FUNCTION_BLOCK FB_System_BWK_931
VAR_INPUT
	Freigabe_auto			: BOOL;
	Betrieb_Anford_auto		: BOOL;
	Regelung_Sollw_auto		: REAL;
END_VAR
VAR_OUTPUT
	{attribute 'OPC.UA.DA' := '1'}Steuerung				: ST_System_BWK_Steuerung;		
	{attribute 'OPC.UA.DA' := '1'}Stellwert				: ST_System_BWK_Stellwert;		
	{attribute 'OPC.UA.DA' := '1'}Zustand					: ST_System_BWK_Zustand;	
	{attribute 'OPC.UA.DA' := '1'}Parameter				: ST_System_BWK_Parameter;		
END_VAR
VAR
	Stellventil_331			: FB_SV;
	Regelventil_331			: FB_RV;
	Brennwertkessel_931		: FB_BWK;

	Zustandscheck			: FB_System_BWK_Zustandscheck;
	Logik					: FB_System_BWK_Logik;
	Ablaufsteuerung			: FB_System_BWK_Ablaufsteuerung;
	Sollwertscheck			: FB_System_BWK_Sollwertscheck;
END_VAR
VAR // added by the converter: edge detectors and wires of the graphical bodies
    _w1, _w2 : ANY;
END_VAR

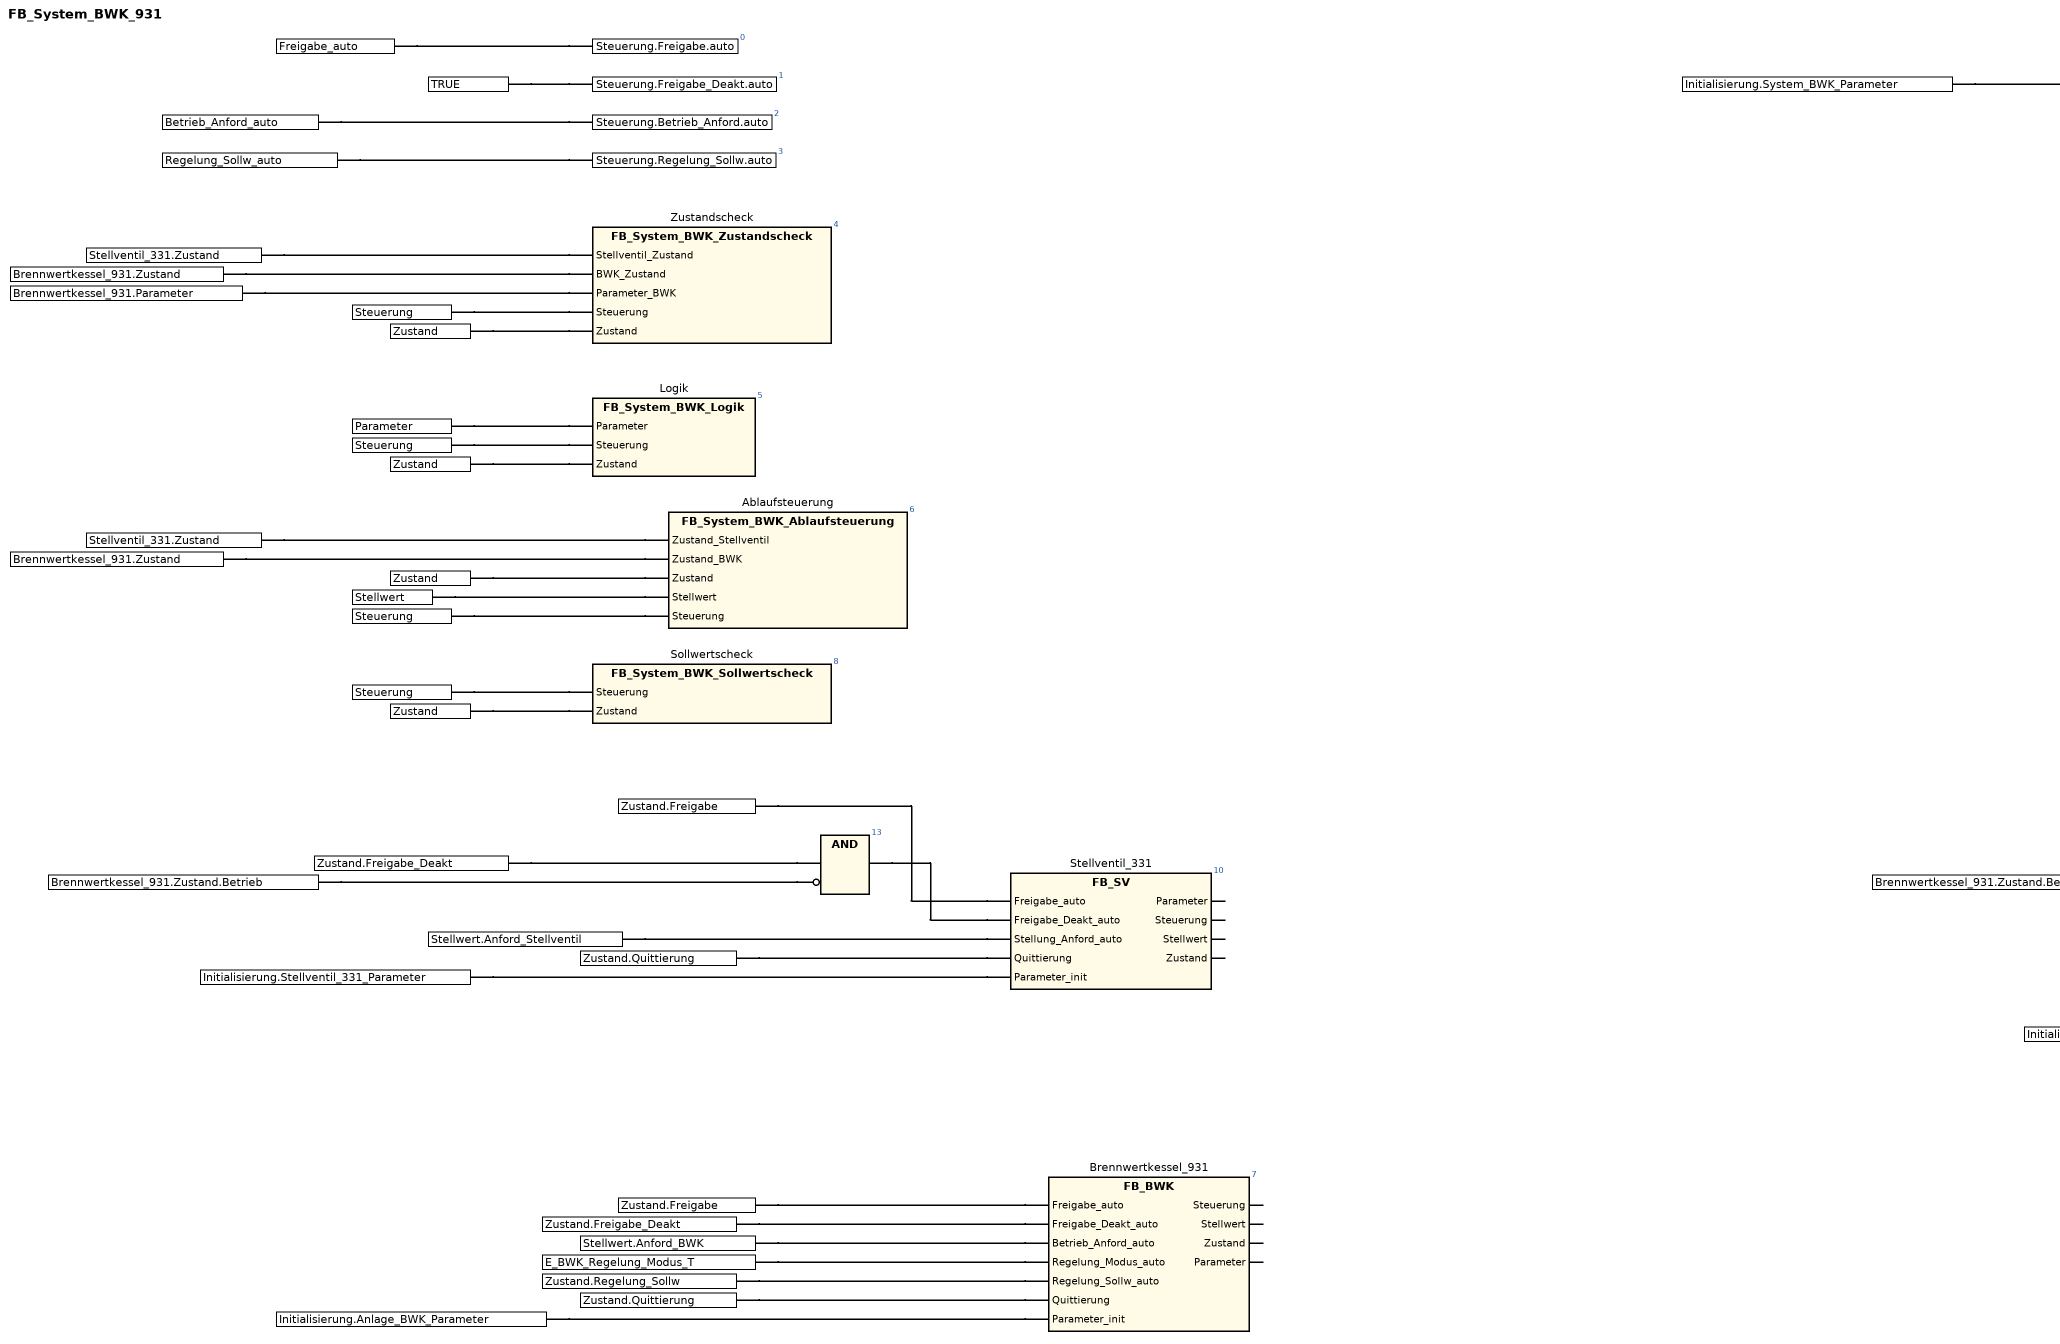
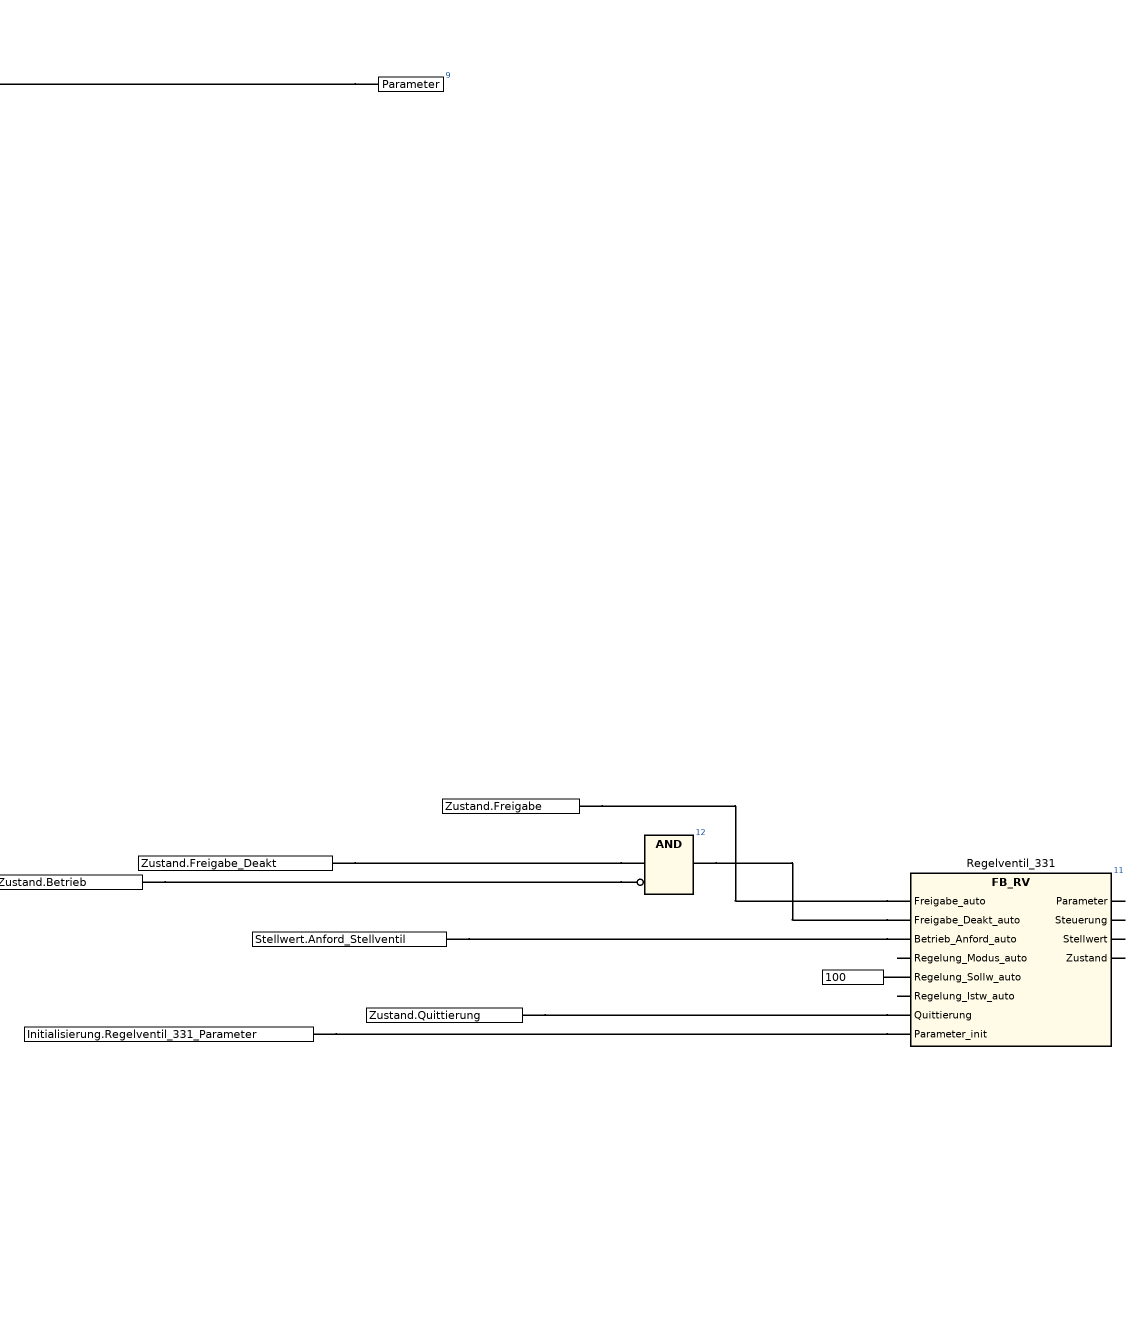
Steuerung.Freigabe.auto := Freigabe_auto;
Steuerung.Freigabe_Deakt.auto := TRUE;
Steuerung.Betrieb_Anford.auto := Betrieb_Anford_auto;
Steuerung.Regelung_Sollw.auto := Regelung_Sollw_auto;
Zustandscheck(
    Stellventil_Zustand := Stellventil_331.Zustand,
    BWK_Zustand := Brennwertkessel_931.Zustand,
    Parameter_BWK := Brennwertkessel_931.Parameter,
    Steuerung := Steuerung,
    Zustand := Zustand); // FB_System_BWK_Zustandscheck
Logik(Parameter := Parameter, Steuerung := Steuerung, Zustand := Zustand); // FB_System_BWK_Logik
Ablaufsteuerung(
    Zustand_Stellventil := Stellventil_331.Zustand,
    Zustand_BWK := Brennwertkessel_931.Zustand,
    Zustand := Zustand,
    Stellwert := Stellwert,
    Steuerung := Steuerung); // FB_System_BWK_Ablaufsteuerung
Brennwertkessel_931(
    Freigabe_auto := Zustand.Freigabe,
    Freigabe_Deakt_auto := Zustand.Freigabe_Deakt,
    Betrieb_Anford_auto := Stellwert.Anford_BWK,
    Regelung_Modus_auto := E_BWK_Regelung_Modus_T,
    Regelung_Sollw_auto := Zustand.Regelung_Sollw,
    Quittierung := Zustand.Quittierung,
    Parameter_init := Initialisierung.Anlage_BWK_Parameter); // FB_BWK
Sollwertscheck(Steuerung := Steuerung, Zustand := Zustand); // FB_System_BWK_Sollwertscheck
Parameter := Initialisierung.System_BWK_Parameter;
Stellventil_331(
    Freigabe_auto := Zustand.Freigabe,
    Freigabe_Deakt_auto := _w1,
    Stellung_Anford_auto := Stellwert.Anford_Stellventil,
    Quittierung := Zustand.Quittierung,
    Parameter_init := Initialisierung.Stellventil_331_Parameter); // FB_SV
Regelventil_331(
    Freigabe_auto := Zustand.Freigabe,
    Freigabe_Deakt_auto := _w2,
    Betrieb_Anford_auto := Stellwert.Anford_Stellventil,
    Regelung_Sollw_auto := 100,
    Quittierung := Zustand.Quittierung,
    Parameter_init := Initialisierung.Regelventil_331_Parameter); // FB_RV
_w2 := Zustand.Freigabe_Deakt AND NOT Brennwertkessel_931.Zustand.Betrieb;
_w1 := Zustand.Freigabe_Deakt AND NOT Brennwertkessel_931.Zustand.Betrieb;

END_FUNCTION_BLOCK

(* stored: Version 1.1.0.1, ProductVersion 3.1.4024.9
   POU FB_System_BWK_931: Id {b46c011f-04fb-49f9-94fb-b0e01fb20880}, SpecialFunc None *)
